// Mitsubishi GX Works2 project: 0710   PLC: Q02/Q02H

PROGRAM MAIN
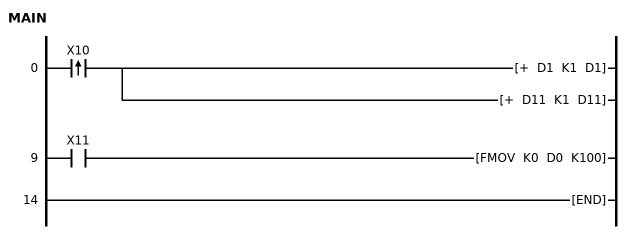
0     LDP     X10
      +       D1 K1 D1
      +       D11 K1 D11
9     LD      X11
      FMOV    K0 D0 K100
14    END
END_PROGRAM

PROGRAM MAIN1
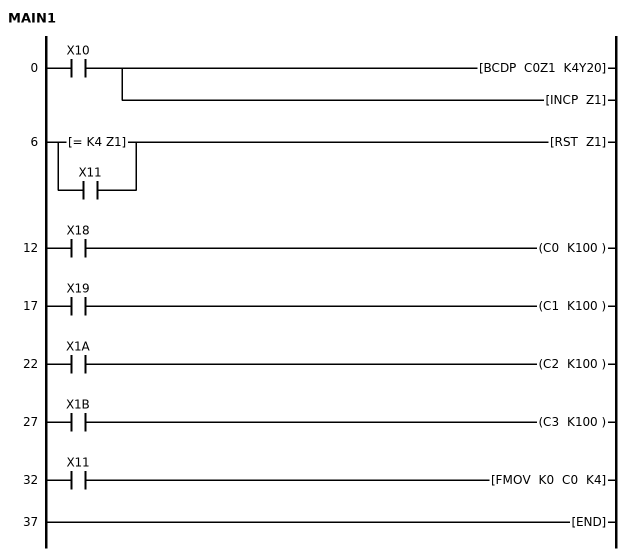
0     LD      X10
      BCDP    C0Z1 K4Y20
      INCP    Z1
6     LD=     K4 Z1
      OR      X11
      RST     Z1
12    LD      X18
      OUT     C0 K100
17    LD      X19
      OUT     C1 K100
22    LD      X1A
      OUT     C2 K100
27    LD      X1B
      OUT     C3 K100
32    LD      X11
      FMOV    K0 C0 K4
37    END
END_PROGRAM

PROGRAM MAIN2
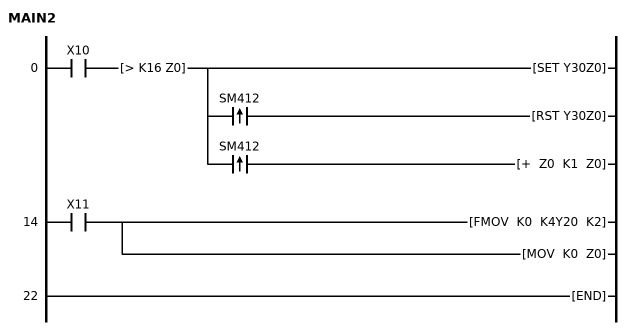
0     LD      X10
      AND>    K16 Z0
      SET     Y30Z0
      MPS
      ANDP    SM412
      RST     Y30Z0
      MPP
      ANDP    SM412
      +       Z0 K1 Z0
14    LD      X11
      FMOV    K0 K4Y20 K2
      MOV     K0 Z0
22    END
END_PROGRAM
